Fanuc KAREL source: d_cmos2sh_c.kl

PROGRAM D_CMOS2SH_C
%NOLOCKGROUP
%CMOSVARS
%CMOS2SHADOW
VAR
	I : INTEGER
	R : REAL
	S : STRING[8]
	P : XYZWPR
	C IN CMOS : INTEGER
	H IN SHADOW : REAL
BEGIN
	I = 1
	R = 2.5
	S = 'abc'
	C = I + 1
	H = R * 2
	WRITE('I = ', I, ' S = ', S, CR)
END D_CMOS2SH_C
